// TIA Portal V19 export
DATA_BLOCK "iDBF_MainSafety"   // DB900, F_DB
NAME : FUSI
// stored: AutoNumber false, InstanceOfName MainSafety, InstanceOfType FB
"MainSafety"
BEGIN
END_DATA_BLOCK
